(* PLC project liner_cyclic.project, CODESYS CODESYS V3.5 SP17 Patch 3 *)
(* stored: creationDateTime 1970-01-01T00:00:00, modificationDateTime 1970-01-01T00:00:00 *)

PROGRAM PLC_PRG

            GVL.PDQ4_F1_PWR_OO := TRUE;  // Подача питания на силовой контактор
GVL.PDQ0_COL_24V := TRUE;    // Подача питания на колонну
Sensors();
SafetyChain();
ServoControl();








          
END_PROGRAM
